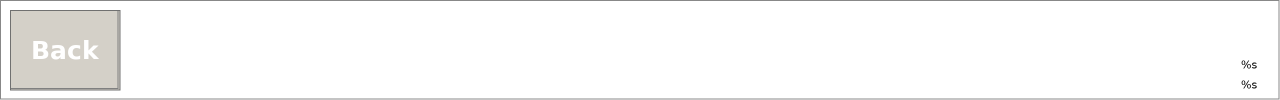
VISUALIZATION Footer_Back  // 1280x100
    Textfield (1160,70 100x30), "%s", text variable: MAIN.fb_TimeStamp.SystemDate
    Textfield (1160,50 100x30), "%s", text variable: MAIN.fb_TimeStamp.SystemTime
    Button (10,10 110x80), "Back"
        OnMouseClick: execute {
            LOGFILE( sLogEvent	 := MSG.EVENT_BTN,
            		 sLogComp	 := MSG.COMP_HMI,
            		 sLogAction	 := MSG.ACTION_BACK,
            	 	 logFlag	 := TRUE);
        }
        OnMouseClick: change screen: PAGE_MAIN
END_VISUALIZATION

(* stored: Version 1.1.0.1, ProductVersion 3.1.4024.12
   Visu Footer_Back: Id {ce661f61-4053-4403-abd3-f1c4aea16582} *)
